(* IEC 61131-3 sources: learning-path/06_oop_in_st/exercises/0_basic_valve_class/src, 3 files *)

(* ---- Tank.st ---- *)
NAMESPACE FluidHandling
    FUNCTION_BLOCK Tank
        VAR_INPUT
            cmdFill: BOOL;
            cmdEmpty: BOOL;
        END_VAR
        VAR_OUTPUT
            inletOpen: BOOL;
            outletOpen: BOOL;
        END_VAR
        VAR
            inlet: Valve;
            outlet: Valve;
        END_VAR

        inlet(cmdOpen := cmdFill,
            ctrlOpen => inletOpen);
        outlet(cmdOpen := cmdEmpty,
                ctrlOpen => outletOpen);
    END_FUNCTION_BLOCK

END_NAMESPACE

(* ---- Valve.st ---- *)
NAMESPACE FluidHandling
    FUNCTION_BLOCK Valve
        VAR_INPUT
            cmdOpen: BOOL;
        END_VAR
        VAR_OUTPUT
            ctrlOpen : BOOL;
            isOpen : BOOL;
            isClosed : BOOL;
        END_VAR

        IF (cmdOpen) THEN
            isOpen := TRUE;
            isClosed := FALSE;
            ctrlOpen := TRUE;
        ELSE
            isOpen := FALSE;
            isClosed := TRUE;
            ctrlOpen := FALSE;
        END_IF;

    END_FUNCTION_BLOCK

END_NAMESPACE

(* ---- ValveBase.st ---- *)
//Use the same namespace than the TYPE for the Valves state

NAMESPACE FluidHandlingClass

    CLASS ValveBase
        VAR

        END_VAR

        METHOD PUBLIC Open
            ;
        END_METHOD

        METHOD PUBLIC Close
            ;
        END_METHOD

        METHOD PUBLIC GetState: FluidHandlingClass.ValveState
            ;
        END_METHOD

        METHOD PUBLIC WriteCyclic
            ;
        END_METHOD

    END_CLASS

END_NAMESPACE
